// TIA Portal V20 export
DATA_BLOCK "DB_SystemSSR"   // DB5
// stored: Access Published, MemoryReserve 100, Namespace Global
   VAR
      FromHMI : Struct
         Line : Struct
            ProductionLine : "Global.SystemSSR";
            EmptyLine { S7_SetPoint := 'True'} : "Global.SystemSSR";
            PackedLine { S7_SetPoint := 'True'} : "Global.SystemSSR";
         END_STRUCT;
      END_STRUCT;
      Line : Struct
         ProductionLine : "Global.SystemSSR";
         EmptyLine { S7_SetPoint := 'True'} : "Global.SystemSSR";
         PackedLine { S7_SetPoint := 'True'} : "Global.SystemSSR";
      END_STRUCT;
      Zone : Struct
         "1" : "Global.SystemSSR";
         "2" : "Global.SystemSSR";
      END_STRUCT;
   END_VAR
BEGIN
END_DATA_BLOCK
